// Implicitly generated code : DO NOT EDIT
FUNCTION CheckLRangeUnsigned : ULINT
VAR_INPUT
	value, lower, upper: ULINT;
END_VAR

{noflow}
IF (value < lower) THEN
	CheckRangeUnsigned := lower;
	F_LogLA3(E_LogLevel.eFatal, 'CheckLRangeUnsigned', 'Check ULINT range unsigned exception: {value} {lower} {upper}', value, lower, upper);
ELSIF(value > upper) THEN
	CheckRangeUnsigned := upper;
	F_LogLA3(E_LogLevel.eFatal, 'CheckLRangeUnsigned', 'Check ULINT range unsigned exception: {value} {lower} {upper}', value, lower, upper);
ELSE
	CheckRangeUnsigned := value;
END_IF
{flow}

END_FUNCTION

(* stored: Version 1.1.0.1, ProductVersion 3.1.4024.0
   POU CheckLRangeUnsigned: Id {24816c5e-0e78-410f-bf49-253138128feb}, SpecialFunc CheckLRangeUnsigned *)
